(* CoDeSys 2.3.9.47 project: ATS_P4.pro *)
(* Libraries: STANDARD.LIB 5.6.98 12:03:02 *)

(* Task configuration *)
TASK Standard (PRIORITY := 0, INTERVAL := T#10ms);
	MAIN
END_TASK

(* POU MAIN, ST *)
PROGRAM MAIN
VAR
	w_myWord		: WORD	:= 16#5D7A;
	w_res_myWord	: WORD	;
	(**)
	dw_myDWord		: DWORD	;
	w_testSW		: WORD	:= 16#1D06;
	myFcn			: fcnblk_process_sw;
	b_ovr_err_var	: BOOL	;
	myArray 		: ARRAY[1..10] OF REAL;(*:= 0, 1, 2, 3, 4, 5, 6, 7, 8, 9*)
END_VAR
(*
	Shift right bitwise (SHR)
	3 times -> n/8
*)
w_res_myWord := SHR(w_myWord,3);

(*
	Shift left bitwise (SHL)
	3 times -> n*8
	Save first in DWORD to prevent cut
*)

dw_myDWord := w_myWord;
dw_myDWord := SHL(w_myWord,3);

(*
	Bitwise OR
	Set MSB 0...3 to 1
*)
dw_myDWord := (16#F0000000 OR w_myWord);

(*
	Function Block
	Process Status Word
*)
(*Function Call*)
myFcn();
(*Assign Function Value*)
myFcn.w_sw := w_testSW;
(*Explicite Variable Definition*)
b_ovr_err_var := myFcn.b_overrunErr;

(*Fill single Entry*)
myArray[1] := 0;
END_PROGRAM

(* POU fcnblk_process_sw, ST *)
FUNCTION_BLOCK fcnblk_process_sw
VAR_INPUT
	w_sw	:	WORD;
END_VAR
VAR_OUTPUT
	i_inLen			: INT ;
	b_overrunErr	: BOOL;
	b_famingErr		: BOOL;
	b_parityErr		: BOOL;
	b_bufferFull	: BOOL;
	b_initAccpted	: BOOL;
	b_rcvRequest	: BOOL;
	b_trtAccepted	: BOOL;
END_VAR
VAR
	(*Position set for first Error Flag*)
	w_err_bitmask	: WORD := 16#0040;
END_VAR
(*Write in Length*)
fcnblk_process_sw.i_inLen := SHR(w_sw,8);
(*Evaluate Error Flags*)
fcnblk_process_sw.b_overrunErr	:= (SHR(w_err_bitmask,0) =(SHR(w_err_bitmask,0) AND w_sw));
fcnblk_process_sw.b_famingErr	:= (SHR(w_err_bitmask,1) =(SHR(w_err_bitmask,1) AND w_sw));
fcnblk_process_sw.b_parityErr	:= (SHR(w_err_bitmask,2) =(SHR(w_err_bitmask,2) AND w_sw));
fcnblk_process_sw.b_bufferFull	:= (SHR(w_err_bitmask,3) =(SHR(w_err_bitmask,3) AND w_sw));
fcnblk_process_sw.b_initAccpted	:= (SHR(w_err_bitmask,4) =(SHR(w_err_bitmask,4) AND w_sw));
fcnblk_process_sw.b_rcvRequest	:= (SHR(w_err_bitmask,5) =(SHR(w_err_bitmask,5) AND w_sw));
fcnblk_process_sw.b_trtAccepted	:= (SHR(w_err_bitmask,6) =(SHR(w_err_bitmask,6) AND w_sw));
END_FUNCTION_BLOCK
